// TwinCAT 3 PLC project Untitled1
// ProgramVersion: 3.1.4024.0
// libraries:
//   Tc2_Standard, * (Beckhoff Automation GmbH)
//   Tc2_System, * (Beckhoff Automation GmbH)
//   Tc3_EventLogger, * (Beckhoff Automation GmbH)
//   Tc3_Module, * (Beckhoff Automation GmbH)
// project tree:
//   / PlcTask.TcTTO
//   POUs/ Class Diagram.TcCD (not stored), MAIN.TcPOU
//   POUs/Module/ FB_Module.TcPOU, I_Module.TcIO
//   POUs/Visitors/ FB_LogCounterValue.TcPOU, FB_LogName.TcPOU, I_VisitModules.TcIO
// real-time tasks:
//   TASK PlcTask: cycle T#10ms, priority 20, ADS port 350

CONFIGURATION Untitled1
    RESOURCE PLC ON TwinCAT3
        TASK PlcTask(INTERVAL := T#10ms, PRIORITY := 20);
        PROGRAM MAIN WITH PlcTask : MAIN;
    END_RESOURCE
END_CONFIGURATION

// ---- POUs/Module/I_Module.TcIO
INTERFACE I_Module

PROPERTY CounterValue : UDINT
GET
END_GET
SET
END_SET
END_PROPERTY

PROPERTY Name : string
GET
END_GET
SET
END_SET
END_PROPERTY

END_INTERFACE

// ---- POUs/Visitors/I_VisitModules.TcIO
INTERFACE I_VisitModules

METHOD VisitModules
VAR_INPUT
	Module : I_Module;
END_VAR
END_METHOD

END_INTERFACE

// ---- POUs/MAIN.TcPOU
PROGRAM MAIN
VAR
	//Modules
	Module_One : FB_Module;
	Module_Two : FB_Module;

	//Visitors
	LogName			: FB_LogName;
	LogCounterValue : FB_LogCounterValue;

	//Test Vars
	writeToLog : BOOL;
END_VAR

Module_One.Name := 'Module One';
Module_Two.Name := 'Module Two';

//
IF writeToLog THEN
	writeToLog := FALSE;
	Module_One.Accept(Visitor := LogName);
	Module_Two.Accept(Visitor := LogName);
END_IF

Module_One.CyclicLogic();
Module_Two.CyclicLogic();

//
IF Module_One.CounterValue = 10 THEN
	Module_Two.Accept(Visitor := LogCounterValue);
END_IF

END_PROGRAM

// ---- POUs/Module/FB_Module.TcPOU
FUNCTION_BLOCK FB_Module IMPLEMENTS I_Module
VAR
	_Name : STRING;
	_Counter : udint;
END_VAR

METHOD Accept
VAR_INPUT
	Visitor : I_VisitModules;
END_VAR
Visitor.VisitModules(THIS^);
END_METHOD

PROPERTY CounterValue : UDINT
GET
CounterValue := _Counter;
END_GET
SET
_Counter := CounterValue;
END_SET
END_PROPERTY

METHOD CyclicLogic : BOOL
VAR_INPUT
END_VAR
_Counter := _Counter + 1;
END_METHOD

PROPERTY Name : STRING
GET
Name := _Name;
END_GET
SET
_Name := NAme;
END_SET
END_PROPERTY

END_FUNCTION_BLOCK

// ---- POUs/Visitors/FB_LogName.TcPOU
FUNCTION_BLOCK FB_LogName IMPLEMENTS I_VisitModules
VAR
END_VAR

METHOD VisitModules
VAR_INPUT
	Module	: I_Module;
END_VAR
ADSLOGSTR(ADSLOG_MSGTYPE_HINT OR ADSLOG_MSGTYPE_LOG, 'The Module Name is: %s', Module.Name);
END_METHOD

END_FUNCTION_BLOCK

// ---- POUs/Visitors/FB_LogCounterValue.TcPOU
FUNCTION_BLOCK FB_LogCounterValue IMPLEMENTS I_VisitModules
VAR_INPUT
END_VAR
VAR_OUTPUT
END_VAR
VAR
END_VAR

METHOD VisitModules
VAR_INPUT
	Module	: I_Module;
END_VAR
ADSLOGDINT(ADSLOG_MSGTYPE_HINT OR ADSLOG_MSGTYPE_LOG, 'The Module Counter is: %d', Module.CounterValue);
END_METHOD

END_FUNCTION_BLOCK
